// TIA Portal V20 export
DATA_BLOCK "ControlNodes"   // DB102
// stored: MemoryReserve 100, Namespace Unit1.Em10
   VAR
      em : "LAF_typeEmControlNode";
      emstate { S7_SetPoint := 'True'} : "LUC_typeStates";
      cm : "Unit1.Em10.typeCmControlNode";
      citiMap : Struct
         PMC : "LER_PMC_Input_Data";
         FlexNet { S7_SetPoint := 'True'} : "LER_FlexNet_Data";
      END_STRUCT;
      laserMark : "Unit1.Em10.typeSequenceControlNode";
      emData : "LER_typePartData";
      SpecialFunctionMode : Struct
         DryRun : Struct
            JRdetectPV : Array[0..15] of Bool;
         END_STRUCT;
      END_STRUCT;
      cmLaserMarkJRDetect : "LBC_typeDigitalSignalControlNode";
      cmLaserMarkStageLiftUpDown : "LBC_typeTwoWayActuatorControlNode";
      cmLaserMarkCoverUpDown : "LBC_typeTwoWayActuatorControlNode";
      cmLaserMarkControl : "LER_typeLaserMarkControlNode";
      cmQrFixReaderControl : "LER_typeSRX300ControlNode";
      GenerateComplete_1 : Bool;
      GenerateComplete_2 : Bool;
   END_VAR
BEGIN
END_DATA_BLOCK
